PROGRAM EM02_Shuttle
VAR
END_VAR

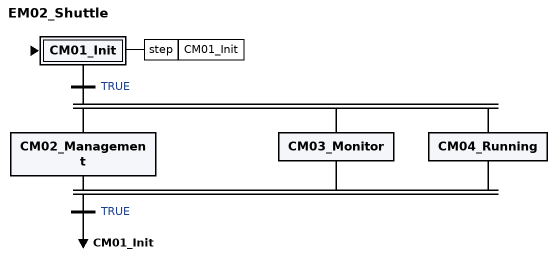
INITIAL_STEP CM01_Init:
    CM01_Init(N);  // step action
END_STEP
TRANSITION FROM CM01_Init TO (CM02_Management, CM03_Monitor, CM04_Running)
    := TRUE;
END_TRANSITION
STEP CM02_Management:
END_STEP
STEP CM03_Monitor:
END_STEP
STEP CM04_Running:
END_STEP
TRANSITION FROM (CM02_Management, CM03_Monitor, CM04_Running) TO CM01_Init
    := TRUE;
END_TRANSITION

ACTION CM01_Init:

END_ACTION

ACTION CM02_Management:
// NETWORK 1
END_ACTION

ACTION CM03_Monitor:
// NETWORK 1
END_ACTION

ACTION CM04_Running:
// NETWORK 1
END_ACTION

END_PROGRAM

(* stored: Version 1.1.0.1, ProductVersion 3.1.4024.9
   POU EM02_Shuttle: Id {20934305-ab74-4a6d-b2df-eb084b1de1c8}, SpecialFunc None
   Action CM01_Init: Id {8fdf3d24-1827-419e-b9c4-ef48af967eb8}
   Action CM02_Management: Id {f28d58db-3dec-40ec-83fa-246276894730}
   Action CM03_Monitor: Id {623e0437-2281-4b46-b59d-614c3f7bc9a5}
   Action CM04_Running: Id {2aa8ca03-9f39-45fa-be62-ba75c00d5f94} *)
